(* CoDeSys 2.3 export: CONTROL_CARRITOS.EXP *)

(* POU Automatico/Exterior/Control_AGV/Control_carritos, LD *)
FUNCTION_BLOCK Control_carritos
VAR_INPUT
	Sensor: BOOL;
	Almacen:BOOL;
	I: BOOL;
	Espera: BOOL;
	Carga:BOOL;
	E:BOOL;
END_VAR
VAR_OUTPUT
	Aviso: BOOL;
	Motor_AV: BOOL;
	Motor_RE: BOOL;

END_VAR
VAR
	E0: BOOL;
	E1: BOOL;

	E2: BOOL;

	E3: BOOL;
	E4: BOOL;

	E5: BOOL;
	E6: BOOL;
	Eaux:BOOL;
	AT2: BOOL;
	FT2:BOOL;

	Carrito_cargado: F_TRIG;
	Temp:TON;
END_VAR
VAR (* helpers for the ST form of the networks *)
	_p1 : BOOL;
	_p2 : BOOL;
	_p3 : BOOL;
	_p4 : BOOL;
	_p5 : BOOL;
	_p6 : BOOL;
END_VAR
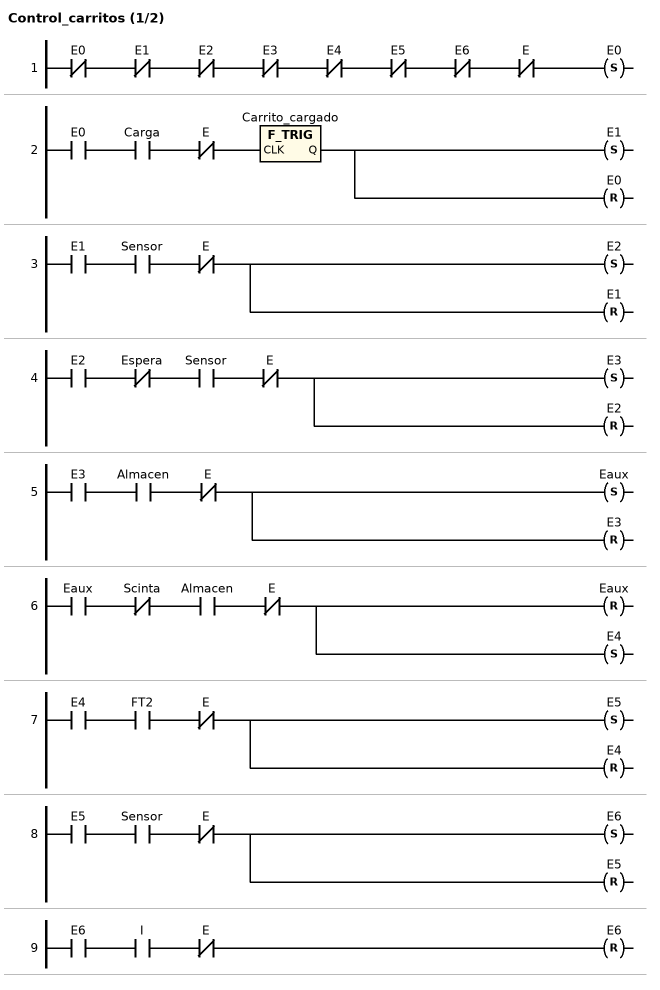
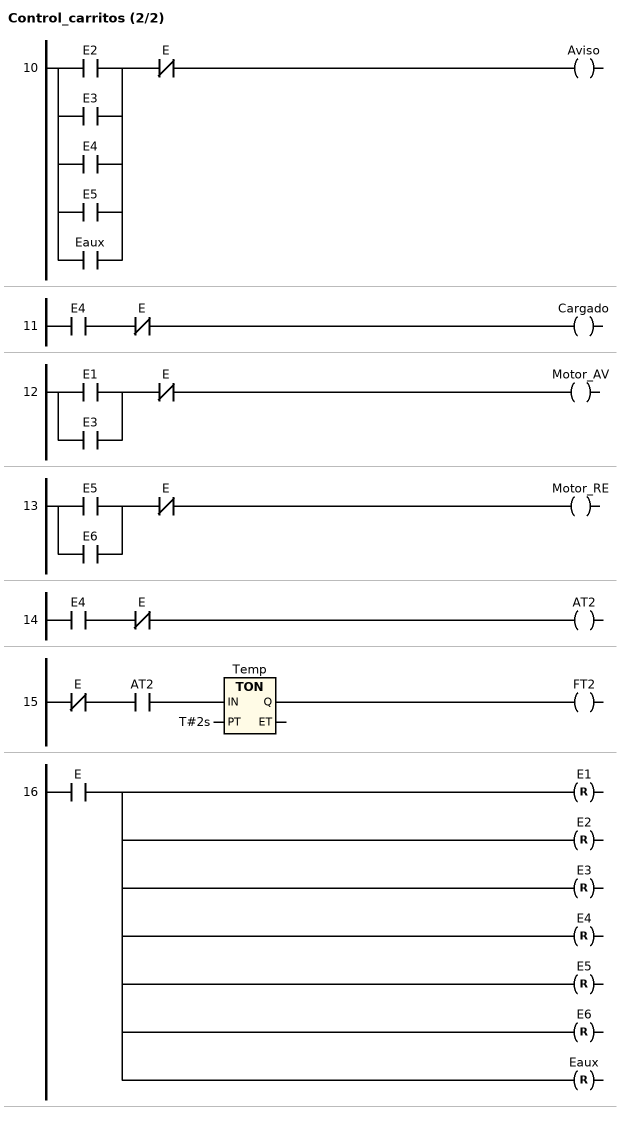
_LD_ (* Ladder Diagram *)
NETWORK 1
	[/E0] - [/E1] - [/E2] - [/E3] - [/E4] - [/E5] - [/E6] - [/E] --- (S E0)
NETWORK 2
	[E0] - [Carga] - [/E] - Carrito_cargado:F_TRIG(CLK: *) --- (S E1) (R E0)
NETWORK 3
	[E1] - [Sensor] - [/E] --- (S E2) (R E1)
NETWORK 4
	[E2] - [/Espera] - [Sensor] - [/E] --- (S E3) (R E2)
NETWORK 5
	[E3] - [Almacen] - [/E] --- (S Eaux) (R E3)
NETWORK 6
	[Eaux] - [/Scinta] - [Almacen] - [/E] --- (R Eaux) (S E4)
NETWORK 7
	[E4] - [FT2] - [/E] --- (S E5) (R E4)
NETWORK 8
	[E5] - [Sensor] - [/E] --- (S E6) (R E5)
NETWORK 9
	[E6] - [I] - [/E] --- (R E6)
NETWORK 10
	{ [E2] | [E3] | [E4] | [E5] | [Eaux] } - [/E] --- (Aviso)
NETWORK 11
	[E4] - [/E] --- (Cargado)
NETWORK 12
	{ [E1] | [E3] } - [/E] --- (Motor_AV)
NETWORK 13
	{ [E5] | [E6] } - [/E] --- (Motor_RE)
NETWORK 14
	[E4] - [/E] --- (AT2)
NETWORK 15
	[/E] - [AT2] - Temp:TON(IN: *, PT: T#2s) --- (FT2)
NETWORK 16
	[E] --- (R E1) (R E2) (R E3) (R E4) (R E5) (R E6) (R Eaux)
_END_LD_
(* the same logic as Structured Text *)
(* Network 1 *)
IF NOT E0 AND NOT E1 AND NOT E2 AND NOT E3 AND NOT E4 AND NOT E5 AND NOT E6 AND NOT E THEN E0 := TRUE; END_IF;
(* Network 2 *)
Carrito_cargado(CLK := E0 AND Carga AND NOT E);
IF Carrito_cargado.Q THEN E1 := TRUE; E0 := FALSE; END_IF;
(* Network 3 *)
_p1 := E1 AND Sensor AND NOT E;
IF _p1 THEN E2 := TRUE; E1 := FALSE; END_IF;
(* Network 4 *)
_p2 := E2 AND NOT Espera AND Sensor AND NOT E;
IF _p2 THEN E3 := TRUE; E2 := FALSE; END_IF;
(* Network 5 *)
_p3 := E3 AND Almacen AND NOT E;
IF _p3 THEN Eaux := TRUE; E3 := FALSE; END_IF;
(* Network 6 *)
_p4 := Eaux AND NOT Scinta AND Almacen AND NOT E;
IF _p4 THEN Eaux := FALSE; E4 := TRUE; END_IF;
(* Network 7 *)
_p5 := E4 AND FT2 AND NOT E;
IF _p5 THEN E5 := TRUE; E4 := FALSE; END_IF;
(* Network 8 *)
_p6 := E5 AND Sensor AND NOT E;
IF _p6 THEN E6 := TRUE; E5 := FALSE; END_IF;
(* Network 9 *)
IF E6 AND I AND NOT E THEN E6 := FALSE; END_IF;
(* Network 10 *)
Aviso := (E2 OR E3 OR E4 OR E5 OR Eaux) AND NOT E;
(* Network 11 *)
Cargado := E4 AND NOT E;
(* Network 12 *)
Motor_AV := (E1 OR E3) AND NOT E;
(* Network 13 *)
Motor_RE := (E5 OR E6) AND NOT E;
(* Network 14 *)
AT2 := E4 AND NOT E;
(* Network 15 *)
Temp(IN := NOT E AND AT2, PT := T#2s);
FT2 := Temp.Q;
(* Network 16 *)
IF E THEN E1 := FALSE; E2 := FALSE; E3 := FALSE; E4 := FALSE; E5 := FALSE; E6 := FALSE; Eaux := FALSE; END_IF;
END_FUNCTION_BLOCK
